# EPICS substitutions: threadExampleApp/Db/user.substitutions
# SPDX-FileCopyrightText: 2006 Argonne National Laboratory
#
# SPDX-License-Identifier: EPICS

# Example substitutions file

file "db/circle.db" {
    { user = "ahdo1293" }
}

file "db/dbExample1.db" {
    { user = "ahdo1293" }
}

file db/dbExample2.db {
    pattern { user, no, scan }
        { "ahdo1293", 1, "1 second" }
        { "ahdo1293", 2, "2 second" }
        { "ahdo1293", 3, "5 second" }
}
